FUNCTION_BLOCK FIELDBUS_ULINT_TO_SIGNAL (* Mirrors IN->OUT if Signal Valid. *)
  (* Standard: 61499-1; Description: Copyright (c) 2026 HR Agrartechnik GmbH This program and the accompanying materials are made available under the terms of the Eclipse Public License 2.0 which is available at https://www.eclipse.org/legal/epl-2.0/ SPDX-License-Identifier: EPL-2.0 *)
  (* Version 1.0, 2026-05-31, Franz Höpfinger, HR Agrartechnik GmbH *)
  PACKAGE logiBUS::signalprocessing::fieldbus;
  IMPORT eclipse4diac::signalprocessing::FIELDBUS_SIGNAL::NOT_AVAILABLE_LWM;
  IMPORT eclipse4diac::signalprocessing::FIELDBUS_SIGNAL::VALID_SIGNAL_LW;
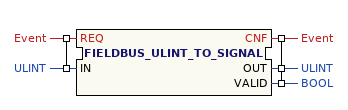
  EVENT_INPUT
    REQ WITH IN; (* Normal Execution Request *)
  END_EVENT
  EVENT_OUTPUT
    CNF WITH OUT, VALID; (* Execution Confirmation *)
  END_EVENT
  VAR_INPUT
    IN : ULINT := LWORD_TO_ULINT(NOT_AVAILABLE_LWM); (* Input *)
  END_VAR
  VAR_OUTPUT
    OUT : ULINT := 16#0000000000000000; (* Output Filtered *)
    VALID : BOOL := FALSE; (* TRUE if Signal is VALID *)
  END_VAR
  EC_STATES
    REQ : REQ -> CNF;
  END_STATES
  ALGORITHM REQ IN ST: (* Executed algorithm *)
IF (IN <= LWORD_TO_ULINT(VALID_SIGNAL_LW)) THEN
	OUT := IN;
	VALID := BOOL#TRUE;
ELSE
	OUT := ULINT#0;
	VALID := BOOL#FALSE;
END_IF;
  END_ALGORITHM
END_FUNCTION_BLOCK
